ABB RobotStudio station: sensor-based-pick-and-place.rsstn

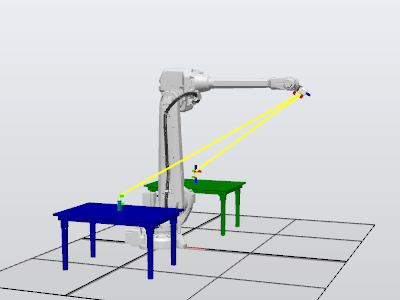
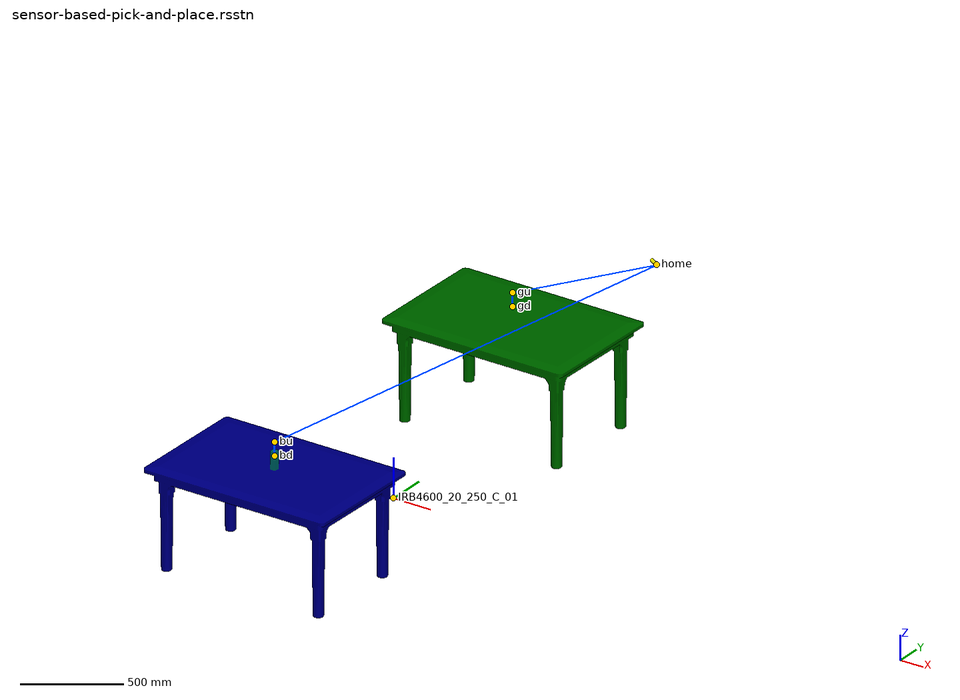
[picture v1: parts stored in the station drawn from their meshes, with robot base, taught points and paths (robot models come from the ABB library and are not in the file)]
Station JawBreaker (saved by RobotStudio 24.3.10885.0)
Controller Controller3
  mechanical unit ROB_1: IRB4600_20_250_C_01, 6 joints, base frame (0, 0, 0) mm
Layout (positions relative to the parent item):
  - IRB4600_20_250_C_01 [mechanism, from %ABB.RobotStudio.Models.IRB4600%\IRB4600_20_250_C_G_01.rslib] at (0, 0, 0) mm; joint values [0, 0, 0, 0, 0.5236, 0] (rad or m)
  - Jaw [mechanism] at (1479.11, 0, 1722.5) mm, rotated rx 180 ry 60 rz 180 deg; joint values [0.02, 0.02] (rad or m)
      TCP Jaw_Tool at (0, 70, 0) mm, rotated rx -90 ry 0 rz 0 deg
      links: L1, L2, L3
  - table2 [part] at (596.07, -724.08, 32.61) mm, rotated rx 90 ry 0 rz 90 deg, size 708.6 x 555.1 x 1062.9 mm
  - table2_2 [part] at (596.07, 1275.92, 32.61) mm, rotated rx 90 ry 0 rz 90 deg, size 708.6 x 555.1 x 1062.9 mm
  - LineSensor [smart component, from Components\LineSensor.rslib] at (1513.75, 0, 1702.5) mm, rotated rx 180 ry 60 rz 180 deg
      properties: Start=[0 0 0]; End=[0 0 0.025]; Length=0.025; Radius=0.01; Tag=(none); SensedPart=(none); SensedPoint=[0 0 0]
    - _sensorPart_ [part], size 20 x 20 x 25 mm
  - Attacher [smart component, from Components\Attacher.rslib]
      properties: Parent=IRB4600_20_250_C_01; Flange=0; Child=(none); Mount=false; Offset=[0 0 0]; Orientation=[0 0 0]
  - Detacher [smart component, from Components\Detacher.rslib]
      properties: Child=(none); KeepPosition=true
  - Part_3 [part] at (15, -1015, 554.71) mm, rotated rx 0 ry 0 rz 90 deg, size 30 x 30 x 100 mm
  - PoseMover [smart component, from Components\PoseMover.rslib]
      properties: Mechanism=Jaw; Pose=3; Duration=0
  - PoseMover_2 [smart component, from Components\PoseMover.rslib]
      properties: Mechanism=Jaw; Pose=2; Duration=0
Attachment: Jaw is attached to IRB4600_20_250_C_01 / Link6
Attachment: LineSensor is attached to Jaw / L1
EventTableEntry 2414: Group=, Trigger=Jaw_signal 2415, Actions=[EventTableActionMechanicalPose 2416], Comment=, ActivationMode=2, Cyclic=false
EventTableTriggerIO 2415: IOValue=[1], IRC5Controller=? -1, Operator=0, SignalSource=Controller3 2422
EventTableActionMechanicalPose 2416: VirtualSignal=, Mechanism=Jaw 2404, ToPoseName=Jaw_opened, VirtualSignalValue=[1]
EventTableEntry 2417: Group=, Trigger=Jaw_signal 2418, Actions=[EventTableActionMechanicalPose 2419], Comment=, ActivationMode=2, Cyclic=false
EventTableTriggerIO 2418: IOValue=[0], IRC5Controller=? -1, Operator=0, SignalSource=Controller3 2422
EventTableActionMechanicalPose 2419: VirtualSignal=, Mechanism=Jaw 2404, ToPoseName=HomePosition, VirtualSignalValue=[1]
EventTableTriggerIO 3531: IOValue=[1], IRC5Controller=? -1, Operator=0, SignalSource=Controller3 2422
EventTableTriggerIO 3532: IOValue=[0], IRC5Controller=? -1, Operator=0, SignalSource=Controller3 2422
Collision set CollisionSet_1:  against , near miss 0 m
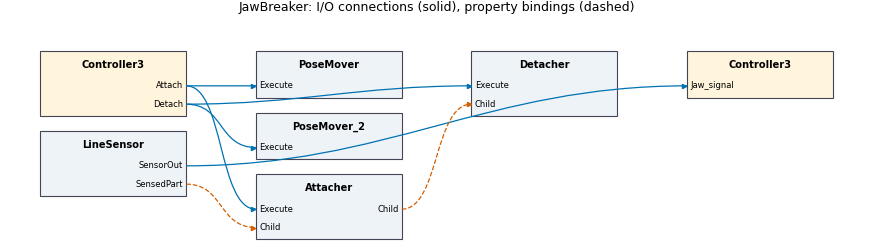
Station logic (signal -> signal, property => property):
  Controller3.Attach -> Attacher.Execute
  Controller3.Detach -> Detacher.Execute
  Controller3.Attach -> PoseMover.Execute
  Controller3.Detach -> PoseMover_2.Execute
  LineSensor.SensorOut -> Controller3.Jaw_signal
  LineSensor.SensedPart => Attacher.Child
  Attacher.Child => Detacher.Child
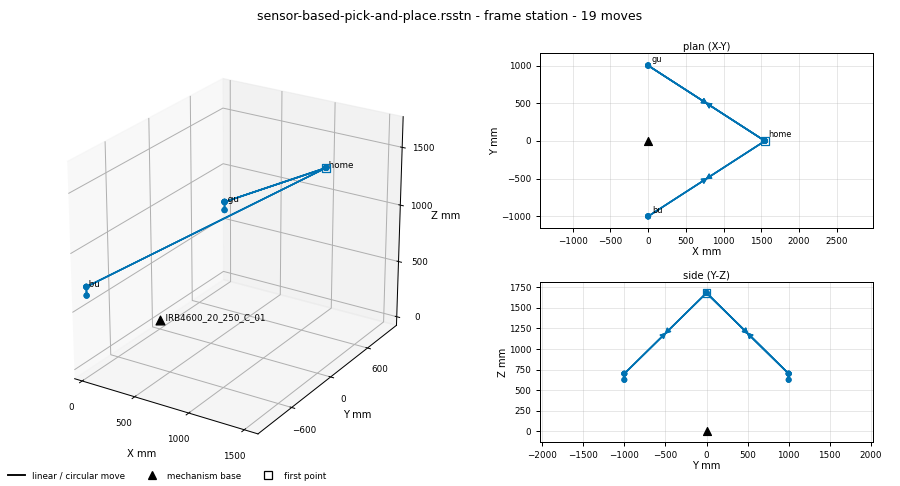
[picture p0: tool path of sensor-based-pick-and-place.rsstn in frame station, 19 of 19 moves have a stored position in this frame; points joined in program order, loops and branches not executed]
Targets, tools, work objects and paths stored in the station, written as RAPID:
! task T_ROB1
MODULE CalibData
  PERS tooldata Jaw_Tool:=[TRUE,[[0,0,80],[1,0,0,0]],[1,[0,0,1],[1,0,0,0],0,0,0]];
  TASK PERS wobjdata mytable:=[FALSE,TRUE,"",[[0,1000,700],[1,0,0,0]],[[0,0,0],[1,0,0,0]]];
ENDMODULE

! task T_ROB1
MODULE Module1
  CONST robtarget gu:=[[-0.000043711,0.000035878,-0.000037534],[-0.000000011,0.707106797,-0.707106766,-0.000000011],[1,0,-1,0],[9E+09,9E+09,9E+09,9E+09,9E+09,9E+09]];
  CONST robtarget gd:=[[-0.000037728,0.000022127,-75.000164328],[0.000000016,-0.707106781,0.707106781,-0.00000001],[1,-1,0,0],[9E+09,9E+09,9E+09,9E+09,9E+09,9E+09]];
  CONST robtarget bu:=[[-0.000043711,-2000.000035878,-0.000037534],[0.000000011,0.707106797,0.707106766,-0.000000011],[-2,-1,0,0],[9E+09,9E+09,9E+09,9E+09,9E+09,9E+09]];
  CONST robtarget bd:=[[-0.000048792,-2000.000022127,-75.000164328],[-0.000000008,0.707106783,0.707106779,-0.000000014],[-2,-1,-1,0],[9E+09,9E+09,9E+09,9E+09,9E+09,9E+09]];
  CONST robtarget home:=[[1548.394191624,-1000,982.5],[0.5,0,0.866025404,0],[-1,0,-1,0],[9E+09,9E+09,9E+09,9E+09,9E+09,9E+09]];
  PROC Path_10()
    MoveL home,v1000,z100,Jaw_Tool\WObj:=mytable;
    MoveL gu,v1000,fine,Jaw_Tool\WObj:=mytable;
    MoveL gd,v1000,fine,Jaw_Tool\WObj:=mytable;
    WaitTime 1;
    MoveL gu,v1000,fine,Jaw_Tool\WObj:=mytable;
    MoveL home,v1000,z100,Jaw_Tool\WObj:=mytable;
    MoveL bu,v1000,fine,Jaw_Tool\WObj:=mytable;
    MoveL bd,v1000,fine,Jaw_Tool\WObj:=mytable;
    PulseDO Detach;
    WaitTime 1;
    MoveL bu,v1000,fine,Jaw_Tool\WObj:=mytable;
    MoveL home,v1000,z100,Jaw_Tool\WObj:=mytable;
    MoveL gu,v1000,fine,Jaw_Tool\WObj:=mytable;
    MoveL home,v1000,z100,Jaw_Tool\WObj:=mytable;
    MoveL bu,v1000,fine,Jaw_Tool\WObj:=mytable;
    MoveL bd,v1000,fine,Jaw_Tool\WObj:=mytable;
    PulseDO Attach;
    WaitTime 1;
    MoveL bu,v1000,fine,Jaw_Tool\WObj:=mytable;
    MoveL home,v1000,z100,Jaw_Tool\WObj:=mytable;
    MoveL gu,v1000,fine,Jaw_Tool\WObj:=mytable;
    MoveL gd,v1000,fine,Jaw_Tool\WObj:=mytable;
    PulseDO Detach;
    WaitTime 1;
    MoveL gu,v1000,fine,Jaw_Tool\WObj:=mytable;
    MoveL home,v1000,z100,Jaw_Tool\WObj:=mytable;
    PulseDO Attach;
  ENDPROC
  PROC main()
    Path_10;
  ENDPROC
ENDMODULE

! task T_ROB1
MODULE user
  TASK PERS wobjdata table:=[FALSE,TRUE,"",[[0,0,0],[1,0,0,0]],[[0,0,0],[1,0,0,0]]];
ENDMODULE

